FUNCTION_BLOCK EL2722
VAR
	{attribute addProperty Name "WcState"}
	_wcState : WcStateBase;
	{attribute addProperty Name "Info data"}
	_infoData : InfoDataBase;
	_io : EL2xx2_Data;
END_VAR

PROPERTY IO : REFERENCE TO EL2xx2_Data
GET
IO REF= _io;
END_GET
END_PROPERTY

PROPERTY WcState : REFERENCE TO WcStateBase
GET
WcState REF= _wcState;
END_GET
END_PROPERTY

END_FUNCTION_BLOCK

(* stored: Version 1.1.0.1, ProductVersion 3.1.4024.9
   POU EL2722: Id {504f799a-c552-0984-30de-22ca18201ec5}, SpecialFunc None
   Property IO: Id {fb1747ef-11c3-02ac-271f-850b74e4abfc}
   Get Get: Id {809601be-ccfa-00a1-2fcd-b50b204a0a4d}
   Property WcState: Id {4b4d91ad-b621-0bf2-21cf-f03e6bcdc1ef}
   Get Get: Id {a68c0116-2158-0f89-037f-ac426a727236} *)
